INTERFACE I_DeserializerArrayForwardEnumerator EXTENDS I_Disposable

PROPERTY PUBLIC Current : I_Deserializer
GET
END_GET
END_PROPERTY

PROPERTY Index : DINT
GET
END_GET
END_PROPERTY

PROPERTY IsValid : BOOL
GET
END_GET
END_PROPERTY

METHOD MoveNext : BOOL
VAR_INPUT
END_VAR
END_METHOD

END_INTERFACE

(* stored: Version 1.1.0.1, ProductVersion 3.1.4024.12
   Itf I_DeserializerArrayForwardEnumerator: Id {21d85085-8288-0789-306f-e652413f69a7}
   Property Current: Id {905b7e5a-bccc-0403-116d-de44aa2fb624}
   Get Get: Id {b4e3bd5e-d787-09d5-017a-67308f982388}
   Property Index: Id {1338b9b4-98f8-0d7d-2483-a849e92014e4}
   Get Get: Id {d7b8612a-a8e5-0e61-006b-0cb7b902dbb4}
   Property IsValid: Id {821b291b-9e37-0760-10d3-7b137b4ff6d0}
   Get Get: Id {d132e1cb-e4e7-0eda-3533-042cb560b56a}
   Method MoveNext: Id {f1369a12-1428-0e66-1bf6-1127d229f9d8} *)
